FUNCTION TryConvert_DWORD_TO_LREAL : BOOL
VAR_INPUT
	in : DWORD;
	out : REFERENCE TO LREAL;
END_VAR

out := DWORD_TO_LREAL(in);
TryConvert_DWORD_TO_LREAL := TRUE;

END_FUNCTION

(* stored: Version 1.1.0.1, ProductVersion 3.1.4024.12
   POU TryConvert_DWORD_TO_LREAL: Id {73e2f749-a9dc-4126-b9a9-2659d092875c}, SpecialFunc None *)
